// TIA Portal V16 export
// export: Created 2023-03-29T11:03:25.348969Z, ExportSetting WithDefaults, DisplayName Totally Integrated Automation Portal, DisplayVersion V16 Update 6, DisplayName TIA Portal Version Control Interface, DisplayVersion V16 Update 2, DisplayName TIA Portal Openness, DisplayVersion V16 Update 6, DisplayName STEP 7 Professional, DisplayVersion V16 Update 6, DisplayName STEP 7 Safety, DisplayVersion V16, DisplayName WinCC Advanced, DisplayVersion V16 Update 6
DATA_BLOCK "MB_TCP_CLIENT"   // DB86
TITLE = CONECT MODBUS TCP SERVER
{ S7_Optimized_Access := 'FALSE' }
AUTHOR : rtecmer
VERSION : 0.1
// stored: AutoNumber true, DBAccessibleFromOPCUA true, IsOnlyStoredInLoadMemory false, IsWriteProtectedInAS false
   VAR
      MB_Client_Receiving : Struct
         Input : Struct
            req : Bool;
            disconnect : Bool;
            mode : USInt;
            mbDataAddr : UDInt;
            CONNECT_ID : UInt := 2;
            IP_OCTET_1 : USInt;
            IP_OCTET_2 : USInt := 0;
            IP_OCTET_3 : USInt := 0;
            IP_OCTET_4 : USInt := 0;
            IP_PORT : UInt;
            MB_MODE : USInt;
            MB_DATA_ADDR : UDInt;
            DATA_LEN : UInt;
            PORT : UInt;
            InOut : Struct
               done : Bool;
               busy : Bool;
               error : Bool;
               STATUS : Word;
               ERROR_STATUS : Word;
            END_STRUCT;
         END_STRUCT;
         tagsStep : Struct
            "step" : Byte;
         END_STRUCT;
      END_STRUCT;
      MB_Client_Receiving_Time : Struct   // Pobieranie nastaw godzin
         Input : Struct
            req : Bool;
            disconnect : Bool;
            mode : USInt;
            mbDataAddr : UDInt;
            CONNECT_ID : UInt := 2;
            IP_OCTET_1 : USInt;
            IP_OCTET_2 : USInt := 0;
            IP_OCTET_3 : USInt := 0;
            IP_OCTET_4 : USInt := 0;
            IP_PORT : UInt;
            MB_MODE : USInt;
            MB_DATA_ADDR : UDInt;
            DATA_LEN : UInt;
            PORT : UInt;
            InOut : Struct
               done : Bool;
               busy : Bool;
               error : Bool;
               STATUS : Word;
               ERROR_STATUS : Word;
            END_STRUCT;
         END_STRUCT;
         tagsStep : Struct
            "step" : Byte;
         END_STRUCT;
      END_STRUCT;
      MB_Client_Sending : Struct   // instancja konfiguracji klient wysyłanie
         Input : Struct
            req : Bool;
            disconnect : Bool;
            mode : USInt;
            mbDataAddr : UDInt;
            CONNECT_ID : UInt;
            IP_OCTET_1 : USInt;
            IP_OCTET_2 : USInt := 0;
            IP_OCTET_3 : USInt := 0;
            IP_OCTET_4 : USInt := 0;
            IP_PORT : UInt;
            MB_MODE : USInt;
            MB_DATA_ADDR : UDInt;
            DATA_LEN : UInt;
            PORT : UInt;
            InOut : Struct
               done : Bool;
               busy : Bool;
               error : Bool;
               STATUS : Word;
               ERROR_STATUS : Word;
            END_STRUCT;
         END_STRUCT;
         tagsStep : Struct
            "step" : Byte;
         END_STRUCT;
      END_STRUCT;
      MB_Client_Sending_1 : Struct   // instancja konfiguracji klient wysyłanie
         Input : Struct
            req : Bool;
            disconnect : Bool;
            mode : USInt;
            mbDataAddr : UDInt;
            CONNECT_ID : UInt;
            IP_OCTET_1 : USInt;
            IP_OCTET_2 : USInt := 0;
            IP_OCTET_3 : USInt := 0;
            IP_OCTET_4 : USInt := 0;
            IP_PORT : UInt;
            MB_MODE : USInt;
            MB_DATA_ADDR : UDInt;
            DATA_LEN : UInt;
            PORT : UInt;
            InOut : Struct
               done : Bool;
               busy : Bool;
               set_step_17 { ExternalAccessible := 'False'; ExternalVisible := 'False'; ExternalWritable := 'False'} : Bool;   // bit inicjacji wysłąnia nowej wartości
               error : Bool;
               STATUS : Word;
               ERROR_STATUS : Word;
            END_STRUCT;
         END_STRUCT;
         tagsStep : Struct
            "step" : Byte;
         END_STRUCT;
      END_STRUCT;
      MB_Client_Sending_2 : Struct   // instancja konfiguracji klient wysyłanie
         Input : Struct
            req : Bool;
            disconnect : Bool;
            mode : USInt;
            mbDataAddr : UDInt;
            CONNECT_ID : UInt;
            IP_OCTET_1 : USInt;
            IP_OCTET_2 : USInt := 0;
            IP_OCTET_3 : USInt := 0;
            IP_OCTET_4 : USInt := 0;
            IP_PORT : UInt;
            MB_MODE : USInt;
            MB_DATA_ADDR : UDInt;
            DATA_LEN : UInt;
            PORT : UInt;
            InOut : Struct
               done : Bool;
               busy : Bool;
               error : Bool;
               STATUS : Word;
               ERROR_STATUS : Word;
            END_STRUCT;
         END_STRUCT;
         tagsStep : Struct
            "step" : Byte;
         END_STRUCT;
      END_STRUCT;
      MB_Client_Sending_3 : Struct   // instancja konfiguracji klient wysyłanie
         Input : Struct
            req : Bool;
            disconnect : Bool;
            mode : USInt;
            mbDataAddr : UDInt;
            CONNECT_ID : UInt;
            IP_OCTET_1 : USInt;
            IP_OCTET_2 : USInt := 0;
            IP_OCTET_3 : USInt := 0;
            IP_OCTET_4 : USInt := 0;
            IP_PORT : UInt;
            MB_MODE : USInt;
            MB_DATA_ADDR : UDInt;
            DATA_LEN : UInt;
            PORT : UInt;
            InOut : Struct
               done : Bool;
               busy : Bool;
               error : Bool;
               STATUS : Word;
               ERROR_STATUS : Word;
            END_STRUCT;
         END_STRUCT;
         tagsStep : Struct
            "step" : Byte;
         END_STRUCT;
      END_STRUCT;
      MB_Client_Sending_4 : Struct   // instancja konfiguracji klient wysyłanie
         Input : Struct
            req : Bool;
            disconnect : Bool;
            mode : USInt;
            mbDataAddr : UDInt;
            CONNECT_ID : UInt;
            IP_OCTET_1 : USInt;
            IP_OCTET_2 : USInt := 0;
            IP_OCTET_3 : USInt := 0;
            IP_OCTET_4 : USInt := 0;
            IP_PORT : UInt;
            MB_MODE : USInt;
            MB_DATA_ADDR : UDInt;
            DATA_LEN : UInt;
            PORT : UInt;
            InOut : Struct
               done : Bool;
               busy : Bool;
               error : Bool;
               STATUS : Word;
               ERROR_STATUS : Word;
            END_STRUCT;
         END_STRUCT;
         tagsStep : Struct
            "step" : Byte;
         END_STRUCT;
      END_STRUCT;
      MB_Client_Sending_5 : Struct   // instancja konfiguracji klient wysyłanie
         Input : Struct
            req : Bool;
            disconnect : Bool;
            mode : USInt;
            mbDataAddr : UDInt;
            CONNECT_ID : UInt;
            IP_OCTET_1 : USInt;
            IP_OCTET_2 : USInt := 0;
            IP_OCTET_3 : USInt := 0;
            IP_OCTET_4 : USInt := 0;
            IP_PORT : UInt;
            MB_MODE : USInt;
            MB_DATA_ADDR : UDInt;
            DATA_LEN : UInt;
            PORT : UInt;
            InOut : Struct
               done : Bool;
               busy : Bool;
               error : Bool;
               STATUS : Word;
               ERROR_STATUS : Word;
            END_STRUCT;
         END_STRUCT;
         tagsStep : Struct
            "step" : Byte;
         END_STRUCT;
      END_STRUCT;
      "step" : Byte;
   END_VAR
BEGIN
END_DATA_BLOCK
